(* CODESYS project Heizungssteuerung.project

Project tree, tasks and I/O mapping:
  Device : CODESYS Control for Raspberry Pi, 3S - Smart Software Solutions GmbH, version 3.5.7.0
    application Application
      libraries: Standard, * (System)
      task MainTask (cyclic, interval t#20ms, priority 1) calls PLC_PRG
      program PLC_PRG [CFC]
      function block Temperaturberechnung [ST]
    SoftMotion General Axis Pool
    GPIOs_A_B : GPIOs A/B, 3S - Smart Software Solutions GmbH, version 1.1.1.0
        unmapped channels: digital inputs (GPIO0..GPIO31), digital outputs (GPIO0..GPIO31)
    I²C
    SPI
    Onewire
    Camera device
      <Leer>
    Ethernet : Ethernet, 3S - Smart Software Solutions GmbH, version 3.5.7.0
        settings: IPAddress = [192,168,24,23]; SubnetMask = [255,255,255,0]; GatewayAddress = [192,168,24,1]; MACAddress = [16#B8,16#27,16#EB,16#6B,16#B4,16#D0]; NetworkInterfaceName = 'eth0'; NetworkInterfaceName = "eth0"
      Modbus_TCP_Master : Modbus TCP Master, 3S - Smart Software Solutions GmbH, version 3.5.6.0
        Modbus_TCP_Slave : Modbus TCP Slave, 3S - Smart Software Solutions GmbH, version 3.5.7.0
            settings: Unit-ID = 1; IPAddress = [192, 168, 24, 40]; Channel 0.Function Code = 3; Channel 0.Read Offset = 16#0000; Channel 0.Read Length = 1; Channel 0.Write Offset = 0; Channel 0.Write Length = 0; Channel 0.Cycle Time = 1000
            input  temp1 : WORD  // Channel 0.Channel 0
            unmapped channels: %IW0 Channel 0
        Modbus_TCP_Slave_1 : Modbus TCP Slave, 3S - Smart Software Solutions GmbH, version 3.5.7.0
            settings: Unit-ID = 2; IPAddress = [192, 168, 24, 23]; Channel 1.Function Code = 3; Channel 1.Read Offset = 16#0000; Channel 1.Read Length = 1; Channel 1.Write Offset = 0; Channel 1.Write Length = 0; Channel 1.Cycle Time = 1000
            input  temp2 : WORD  // Channel 1.Channel 1
            unmapped channels: Channel 1
        Modbus_TCP_Slave_2 : Modbus TCP Slave, 3S - Smart Software Solutions GmbH, version 3.5.7.0
            settings: Unit-ID = 3; IPAddress = [192, 168, 24, 17]; Channel 0.Function Code = 16; Channel 0.Read Offset = 0; Channel 0.Read Length = 0; Channel 0.Write Offset = 16#0000; Channel 0.Write Length = 1; Channel 0.Cycle Time = 1000
            output anzeige_temp : WORD  // Channel 0.Channel 0
            unmapped channels: %QW0 Channel 0
*)

// Device/Application/PLC_PRG
PROGRAM PLC_PRG
VAR
	temp_mittelwert: INT;
	Wohnzimmer: temperaturberechnung;
END_VAR

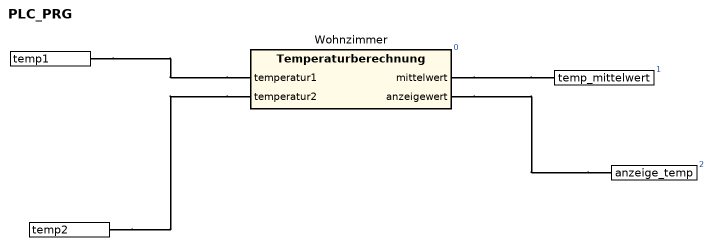
Wohnzimmer(temperatur1 := temp1, temperatur2 := temp2); // Temperaturberechnung
temp_mittelwert := Wohnzimmer.mittelwert;
anzeige_temp := Wohnzimmer.anzeigewert;

END_PROGRAM

// Device/Application/Temperaturberechnung
FUNCTION_BLOCK Temperaturberechnung
VAR_INPUT
	temperatur1: INT;
	temperatur2: INT;
END_VAR
VAR_OUTPUT
	mittelwert: INT;
	anzeigewert: INT;
END_VAR
VAR
END_VAR


mittelwert := (temperatur1 / 10 + temperatur2 / 10) / 2;

anzeigewert := mittelwert * 10;

END_FUNCTION_BLOCK
